INTERFACE ITF_BaseImpulse

END_INTERFACE

(* stored: Version 1.1.0.1
   Itf ITF_BaseImpulse: Id {a073b66d-3394-06c6-376a-ecde61bd42a8} *)
